(* PLC project LibIT_PT, lamsystems-it.ru LibIT_PT 1 *)
(* stored: creationDateTime 2019-11-13T09:37:45, productRelease 0, modificationDateTime 2021-12-27T12:20:59, version 1 *)

(* Установка режима работы входа PT *)
FUNCTION_BLOCK PTMode
  VAR_INPUT
    Ex : BOOL := FALSE;  (* разрешение на выполнение *)
    PTn : BYTE := 0;  (* номер входа *)
    M : BYTE := 0;  (* режим работы *)
    STy : BYTE := 0;  (* тип чувствительного элемента *)
  END_VAR
  VAR_OUTPUT
    Ok : BYTE := 0;  (* код результата исполнения блока *)
  END_VAR

            {extern void App_PTMode(PTMODE*);App_PTMode(data__);}

          
END_FUNCTION_BLOCK

(* Текущий режим и состояние входа PT *)
FUNCTION_BLOCK PTStatus
  VAR_INPUT
    PTn : BYTE := 0;  (* номер входа *)
  END_VAR
  VAR_OUTPUT
    Om : BYTE := 0;  (* режим работы (установленный) *)
    Os : BYTE := 0;  (* код состояния *)
    Ok : BYTE := 0;  (* код результата исполнения блока *)
  END_VAR

            {extern void App_PTStatus(PTSTATUS*);App_PTStatus(data__);}

          
END_FUNCTION_BLOCK

(* Получение значения входа PT *)
FUNCTION_BLOCK PTVal
  VAR_INPUT
    Ex : BOOL := FALSE;  (* разрешение на выполнение *)
    PTn : BYTE := 0;  (* номер входа *)
  END_VAR
  VAR_OUTPUT
    Ov : REAL := 0.0;  (* значение *)
    Ok : BYTE := 0;  (* код результата исполнения блока *)
  END_VAR

            {extern void App_PTVal(PTVAL*);App_PTVal(data__);}

          
END_FUNCTION_BLOCK
